(* PLC project  *)

PROGRAM P
  VAR  (* added by the conversion: wires and edge detectors of the diagram *)
    _AND13_OUT : BOOL;
  END_VAR

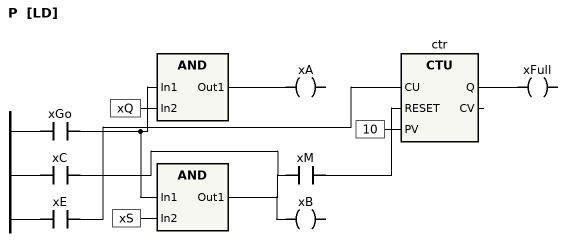
(* LD diagram, written out as Structured Text *)
xA := xGo AND xQ;
_AND13_OUT := xGo AND xS;
xB := _AND13_OUT;
ctr(CU := xE, RESET := (_AND13_OUT OR xC) AND xM, PV := 10);
xFull := ctr.Q;
END_PROGRAM
